// Returns the datatype of a variable as a string using its pointer and size.
// Variables allocated in dynamic memory are not supported.
FUNCTION FsF_GetTypeNameByAddress : FsT_Str
VAR_INPUT
	Address : PVOID; // Pointer to variable.
	Size : FsT_Size; // Size of variable in bytes.
END_VAR
VAR 
	nTmp : UDINT := SIZEOF(FsF_GetTypeNameByAddress);
END_VAR

IF Size = 0 THEN RETURN; END_IF
FsF_IecApplicationInformation().GetDatatypeNameByAddress(TO_UDINT(Size), Address, nTmp, ADR(FsF_GetTypeNameByAddress));

END_FUNCTION

(* stored: Version 1.1.0.1, ProductVersion 3.1.4024.4
   POU FsF_GetTypeNameByAddress: Id {8b0eb9a2-7080-4741-86e4-faa13a477e15}, SpecialFunc None *)
